// Mitsubishi GX Works2 project: 실린더 테스트 동작0912   PLC: Q03UDV

PROGRAM MAIN
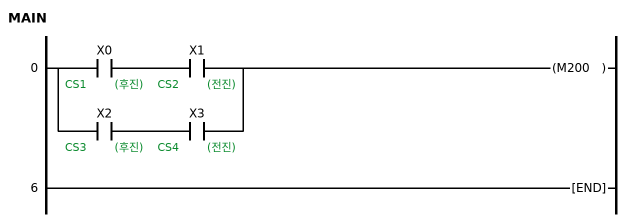
0     LD      X0  ; CS1        (후진)
      AND     X1  ; CS2        (전진)
      LD      X2  ; CS3        (후진)
      AND     X3  ; CS4        (전진)
      ORB
      OUT     M200
6     END
END_PROGRAM

// device comments not shown above
X4  ; 시작
X5  ; 정지
Y10  ; 양솔전진
Y11  ; 양솔후진
Y12  ; 편솔
Y13  ; 부저
